// TIA Portal V21 export
DATA_BLOCK "Paratia"   // DB25
{ S7_Optimized_Access := 'TRUE' }
// stored: MemoryReserve 100
   VAR RETAIN
      P : Array[0.."K_NumParatia"] of "Std_Paratia";
      Posizionamento : Struct
         Paratia : Array[0.."K_NumParatia"] of Struct
            K_Paratia : Int;   // Costante che inidca la paratia
            PosizioneAttuale : Real;   // Posizione attuale della paratia
            Target : Real;   // Quantità che dovrebbe essere gestita
            TargetOld : Real;
            PercentualeDaScarto : Real;   // Percentuale di apertura per compensare lo scarto totale
            PercentualeDaTarget : Real;   // Percentuale di apertura da target
            PercentualeDaGestire : Real;
            OffsetDaPrecedente : Real;   // Posizione offsetta rispetto alla precedente
            Abilitazione : Bool;   // La paratia è abilitata al funzionamento
            StatoAperta : Bool;   // 1 = Aperta 0 = Chiusa
            MassimoProdottoGestibile : Real;
            PulsanteIncrementa_Premuto : Bool;
            PulsanteDecrementa_Premuto : Bool;
            PulsanteIncrementa_Precedente : Bool;
            PulsanteDecrementa_Precedente : Bool;
            Richieste : Struct
               PercProdottoRichiesto : Real;
               QuotaTrovata : Int;
            END_STRUCT;
            Diagnostica : Struct
               MassimoValoreApertura : Bool;
               ParatiaForzataChiusa : Bool;
               TermicoScattato : Bool;
               OvertimeMovimento : Bool;
               SezionatoreAperto : Bool;
               PresaInCaricoDiExtraProdotto : Bool;
               GestioneScartiDisabilitata : Bool;
               ParatiaDisabilitata : Bool;
               ParatiaNonInAutomatico : Bool;
            END_STRUCT;
            VersoLince : Array[0.."K_NumLinci"] of Struct
               PercorsoAttivo : Bool;
               ProdottoOltreMax : Real;
            END_STRUCT;
         END_STRUCT;
         AbilitazioneGestioneScarti : Bool := TRUE;   // Se abilitato lo scarto viene distribuito tra quelle aperte
         EquidistribuzioneCarico : Bool := FALSE;
         Inizializza : Bool := FALSE;
         PercentualeScartata : Real := 0.0;
         PercentualeGestita : Real := 100.0;
         ProdottoAssegnato : Real := 100.0;
         ProdottoNonAssegnato : Real := 0.0;
         NumeroParatieAperte : Int := 2;
         AbilitazioneCalcoloDistribuzione : Bool := TRUE;
         DistribuzioneProdottoNastro : Struct
            Quota : Array[0..99] of Real;   // Quantità di prodotto per ogni quota
         END_STRUCT;
         TargetAutomatico : Bool := TRUE;
      END_STRUCT;
      ProdottoNecessario : Struct
         Lince : Array[0.."K_NumLinci"] of Struct
            ChiamataProdotto : Bool;
            AlimentataDalleParatie : Bool;
            PercentualeAttuale : Real;   // Livello attuale
            PercentualeMassima : Real;   // Livello massimo gestito
            ProdottoRichiestoAssoluto : Real;   // Tiene conto solo della propria chiamata
            ProdottoRichiestoRelativo : Real;   // Tiene conto anche delle altre paratie in chiamata
            ProdottoRichiestoRelativoConExtra : Real;
            ProdottoRichiestoASorgenti : Real;   // Tiene conto del numero di sorgenti collegate
            NumeroSorgentiAttive : Int;
            MassimoProdottoGestibile : Real;
            ProdottoNonGestibile : Real;
            TotaleProdottoExtraTraSorgenti : Real;
         END_STRUCT;
         TotaleRichiesta : Real := 21.65003;
         ProdottoExtraNonGestito : Real := 0.0;
         TotaleRelativoDiChiPuòGestireExtra : Real := 100.0;
      END_STRUCT;
   END_VAR
   VAR
      Funzioni : Struct
         DefaultPrm : Bool := FALSE;
         TutteInAuto : Bool := FALSE;
         PosizionamentiAutomatici : Bool := TRUE;
         BypassFinecorsa : Bool := FALSE;
         VistaLivelloPrograammatore : Bool := FALSE;
      END_STRUCT;
   END_VAR
BEGIN
   // P[0] : Non usare
   // P[1] : IFT6
   // P[2] : IFT7
   // P[3] : IFT8
   // P[4] : IFT9
   // P[5] : Cubettatrice
   // P[6] : Cernita
   P[0].In.SetpointAuto := 0.0;
   P[1].In.SetpointAuto := 100.0;
   P[2].In.SetpointAuto := 34.0;
   P[3..5].In.SetpointAuto := 0.0;
   P[6].In.SetpointAuto := 40.0;
   P[7..9].In.SetpointAuto := 0.0;
   P[0..9].In.PulsanteIncrementa := FALSE;
   P[0..9].In.PulsanteDecrementa := FALSE;
   P[0..9].In.TermicoIntervenuto := FALSE;
   P[0..9].In.FinecorsaPositivo := FALSE;
   P[0..9].In.FinecorsaNegativo := FALSE;
   P[0].In.AbilitazioneMovimento := FALSE;
   P[1..6].In.AbilitazioneMovimento := TRUE;
   P[7..9].In.AbilitazioneMovimento := FALSE;
   P[0].Prm.IsteresiComando := 10.0;
   P[1..2].Prm.IsteresiComando := 6.5;
   P[3..9].Prm.IsteresiComando := 8.0;
   P[0..9].Prm.AbilitazioneInterpolazione := FALSE;
   P[0].Prm.Interpolazione[0].Setpoint := 0.0;
   P[0].Prm.Interpolazione[1].Setpoint := 20.0;
   P[0].Prm.Interpolazione[2].Setpoint := 40.0;
   P[0].Prm.Interpolazione[3].Setpoint := 60.0;
   P[0].Prm.Interpolazione[4].Setpoint := 80.0;
   P[0].Prm.Interpolazione[5].Setpoint := 100.0;
   P[1].Prm.Interpolazione[0].Setpoint := 0.0;
   P[1].Prm.Interpolazione[1].Setpoint := 20.0;
   P[1].Prm.Interpolazione[2].Setpoint := 40.0;
   P[1].Prm.Interpolazione[3].Setpoint := 60.0;
   P[1].Prm.Interpolazione[4].Setpoint := 80.0;
   P[1].Prm.Interpolazione[5].Setpoint := 100.0;
   P[2].Prm.Interpolazione[0].Setpoint := 0.0;
   P[2].Prm.Interpolazione[1].Setpoint := 20.0;
   P[2].Prm.Interpolazione[2].Setpoint := 40.0;
   P[2].Prm.Interpolazione[3].Setpoint := 60.0;
   P[2].Prm.Interpolazione[4].Setpoint := 80.0;
   P[2].Prm.Interpolazione[5].Setpoint := 100.0;
   P[3].Prm.Interpolazione[0].Setpoint := 0.0;
   P[3].Prm.Interpolazione[1].Setpoint := 20.0;
   P[3].Prm.Interpolazione[2].Setpoint := 40.0;
   P[3].Prm.Interpolazione[3].Setpoint := 60.0;
   P[3].Prm.Interpolazione[4].Setpoint := 80.0;
   P[3].Prm.Interpolazione[5].Setpoint := 100.0;
   P[4].Prm.Interpolazione[0].Setpoint := 0.0;
   P[4].Prm.Interpolazione[1].Setpoint := 20.0;
   P[4].Prm.Interpolazione[2].Setpoint := 40.0;
   P[4].Prm.Interpolazione[3].Setpoint := 60.0;
   P[4].Prm.Interpolazione[4].Setpoint := 80.0;
   P[4].Prm.Interpolazione[5].Setpoint := 100.0;
   P[5].Prm.Interpolazione[0].Setpoint := 0.0;
   P[5].Prm.Interpolazione[1].Setpoint := 20.0;
   P[5].Prm.Interpolazione[2].Setpoint := 40.0;
   P[5].Prm.Interpolazione[3].Setpoint := 60.0;
   P[5].Prm.Interpolazione[4].Setpoint := 80.0;
   P[5].Prm.Interpolazione[5].Setpoint := 100.0;
   P[6].Prm.Interpolazione[0].Setpoint := 0.0;
   P[6].Prm.Interpolazione[1].Setpoint := 20.0;
   P[6].Prm.Interpolazione[2].Setpoint := 40.0;
   P[6].Prm.Interpolazione[3].Setpoint := 60.0;
   P[6].Prm.Interpolazione[4].Setpoint := 80.0;
   P[6].Prm.Interpolazione[5].Setpoint := 100.0;
   P[7].Prm.Interpolazione[0].Setpoint := 0.0;
   P[7].Prm.Interpolazione[1].Setpoint := 20.0;
   P[7].Prm.Interpolazione[2].Setpoint := 40.0;
   P[7].Prm.Interpolazione[3].Setpoint := 60.0;
   P[7].Prm.Interpolazione[4].Setpoint := 80.0;
   P[7].Prm.Interpolazione[5].Setpoint := 100.0;
   P[8].Prm.Interpolazione[0].Setpoint := 0.0;
   P[8].Prm.Interpolazione[1].Setpoint := 20.0;
   P[8].Prm.Interpolazione[2].Setpoint := 40.0;
   P[8].Prm.Interpolazione[3].Setpoint := 60.0;
   P[8].Prm.Interpolazione[4].Setpoint := 80.0;
   P[8].Prm.Interpolazione[5].Setpoint := 100.0;
   P[9].Prm.Interpolazione[0].Setpoint := 0.0;
   P[9].Prm.Interpolazione[1].Setpoint := 20.0;
   P[9].Prm.Interpolazione[2].Setpoint := 40.0;
   P[9].Prm.Interpolazione[3].Setpoint := 60.0;
   P[9].Prm.Interpolazione[4].Setpoint := 80.0;
   P[9].Prm.Interpolazione[5].Setpoint := 100.0;
   P[0].Prm.Interpolazione[0].Valore := 0.0;
   P[0].Prm.Interpolazione[1].Valore := 20.0;
   P[0].Prm.Interpolazione[2].Valore := 40.0;
   P[0].Prm.Interpolazione[3].Valore := 60.0;
   P[0].Prm.Interpolazione[4].Valore := 80.0;
   P[0].Prm.Interpolazione[5].Valore := 100.0;
   P[1].Prm.Interpolazione[0].Valore := 0.0;
   P[1].Prm.Interpolazione[1].Valore := 20.0;
   P[1].Prm.Interpolazione[2].Valore := 40.0;
   P[1].Prm.Interpolazione[3].Valore := 60.0;
   P[1].Prm.Interpolazione[4].Valore := 80.0;
   P[1].Prm.Interpolazione[5].Valore := 100.0;
   P[2].Prm.Interpolazione[0].Valore := 0.0;
   P[2].Prm.Interpolazione[1].Valore := 20.0;
   P[2].Prm.Interpolazione[2].Valore := 40.0;
   P[2].Prm.Interpolazione[3].Valore := 60.0;
   P[2].Prm.Interpolazione[4].Valore := 80.0;
   P[2].Prm.Interpolazione[5].Valore := 100.0;
   P[3].Prm.Interpolazione[0].Valore := 0.0;
   P[3].Prm.Interpolazione[1].Valore := 20.0;
   P[3].Prm.Interpolazione[2].Valore := 40.0;
   P[3].Prm.Interpolazione[3].Valore := 60.0;
   P[3].Prm.Interpolazione[4].Valore := 80.0;
   P[3].Prm.Interpolazione[5].Valore := 100.0;
   P[4].Prm.Interpolazione[0].Valore := 0.0;
   P[4].Prm.Interpolazione[1].Valore := 20.0;
   P[4].Prm.Interpolazione[2].Valore := 40.0;
   P[4].Prm.Interpolazione[3].Valore := 60.0;
   P[4].Prm.Interpolazione[4].Valore := 80.0;
   P[4].Prm.Interpolazione[5].Valore := 100.0;
   P[5].Prm.Interpolazione[0].Valore := 0.0;
   P[5].Prm.Interpolazione[1].Valore := 20.0;
   P[5].Prm.Interpolazione[2].Valore := 40.0;
   P[5].Prm.Interpolazione[3].Valore := 60.0;
   P[5].Prm.Interpolazione[4].Valore := 80.0;
   P[5].Prm.Interpolazione[5].Valore := 100.0;
   P[6].Prm.Interpolazione[0].Valore := 0.0;
   P[6].Prm.Interpolazione[1].Valore := 20.0;
   P[6].Prm.Interpolazione[2].Valore := 40.0;
   P[6].Prm.Interpolazione[3].Valore := 60.0;
   P[6].Prm.Interpolazione[4].Valore := 80.0;
   P[6].Prm.Interpolazione[5].Valore := 100.0;
   P[7].Prm.Interpolazione[0].Valore := 0.0;
   P[7].Prm.Interpolazione[1].Valore := 20.0;
   P[7].Prm.Interpolazione[2].Valore := 40.0;
   P[7].Prm.Interpolazione[3].Valore := 60.0;
   P[7].Prm.Interpolazione[4].Valore := 80.0;
   P[7].Prm.Interpolazione[5].Valore := 100.0;
   P[8].Prm.Interpolazione[0].Valore := 0.0;
   P[8].Prm.Interpolazione[1].Valore := 20.0;
   P[8].Prm.Interpolazione[2].Valore := 40.0;
   P[8].Prm.Interpolazione[3].Valore := 60.0;
   P[8].Prm.Interpolazione[4].Valore := 80.0;
   P[8].Prm.Interpolazione[5].Valore := 100.0;
   P[9].Prm.Interpolazione[0].Valore := 0.0;
   P[9].Prm.Interpolazione[1].Valore := 20.0;
   P[9].Prm.Interpolazione[2].Valore := 40.0;
   P[9].Prm.Interpolazione[3].Valore := 60.0;
   P[9].Prm.Interpolazione[4].Valore := 80.0;
   P[9].Prm.Interpolazione[5].Valore := 100.0;
   P[0].Dati.AnalogicaReale := 0.0;
   P[1].Dati.AnalogicaReale := 101.2339;
   P[2].Dati.AnalogicaReale := 34.72675;
   P[3].Dati.AnalogicaReale := 0.0;
   P[4].Dati.AnalogicaReale := 0.4089539;
   P[5].Dati.AnalogicaReale := 0.0;
   P[6].Dati.AnalogicaReale := 45.57193;
   P[7..9].Dati.AnalogicaReale := 0.0;
   P[0].Dati.PosizioneAttuale := 0.0;
   P[1].Dati.PosizioneAttuale := 101.2339;
   P[2].Dati.PosizioneAttuale := 34.72675;
   P[3].Dati.PosizioneAttuale := 0.0;
   P[4].Dati.PosizioneAttuale := 0.4089539;
   P[5].Dati.PosizioneAttuale := 0.0;
   P[6].Dati.PosizioneAttuale := 45.57193;
   P[7..9].Dati.PosizioneAttuale := 0.0;
   P[0].Dati.IncrementaUscita := TRUE;
   P[1..9].Dati.IncrementaUscita := FALSE;
   P[0].Dati.PosizionePrecedente := 0.0;
   P[1].Dati.PosizionePrecedente := 101.0646;
   P[2].Dati.PosizionePrecedente := 24.01413;
   P[3].Dati.PosizionePrecedente := 0.0;
   P[4].Dati.PosizionePrecedente := 10.76733;
   P[5].Dati.PosizionePrecedente := 13.94059;
   P[6].Dati.PosizionePrecedente := 49.32968;
   P[7..9].Dati.PosizionePrecedente := 0.0;
   P[0].Dati.DeltaMovimentoTotale := 0.0;
   P[1].Dati.DeltaMovimentoTotale := 38.55846;
   P[2].Dati.DeltaMovimentoTotale := 95655.14;
   P[3].Dati.DeltaMovimentoTotale := 0.0;
   P[4].Dati.DeltaMovimentoTotale := 276.431;
   P[5].Dati.DeltaMovimentoTotale := 1529.73;
   P[6].Dati.DeltaMovimentoTotale := 26.6803;
   P[7..9].Dati.DeltaMovimentoTotale := 0.0;
   P[0].Dati.DeltaMovimentoTotalePrecedente := 0.0;
   P[1].Dati.DeltaMovimentoTotalePrecedente := 96.96799;
   P[2].Dati.DeltaMovimentoTotalePrecedente := 84.48998;
   P[3].Dati.DeltaMovimentoTotalePrecedente := 0.0;
   P[4].Dati.DeltaMovimentoTotalePrecedente := 6.2173;
   P[5].Dati.DeltaMovimentoTotalePrecedente := 10887.7;
   P[6].Dati.DeltaMovimentoTotalePrecedente := 66.14905;
   P[7..9].Dati.DeltaMovimentoTotalePrecedente := 0.0;
   P[0..9].Dati.VerificaOvertime := FALSE;
   P[0..9].Dati.InAllarme := FALSE;
   P[0..2].Dati.ForzataChiusa := FALSE;
   P[3..4].Dati.ForzataChiusa := TRUE;
   P[5..9].Dati.ForzataChiusa := FALSE;
   P[0..9].Hmi.Auto := TRUE;
   P[0..9].Hmi.Man := FALSE;
   P[0..9].Hmi.PulsanteIncrementa := FALSE;
   P[0..9].Hmi.PulsanteDecrementa := FALSE;
   P[0..9].Hmi.Simulazione := FALSE;
   P[0].Hmi.SetpointBloccato := FALSE;
   P[1..5].Hmi.SetpointBloccato := TRUE;
   P[6..9].Hmi.SetpointBloccato := FALSE;
   P[0..9].Allarmi.TimerRitMov.IN := FALSE;
   P[0..9].Allarmi.TimerRitMov.O := FALSE;
   P[0..9].Allarmi.TimerRitMov.Preset := 5.0;
   P[0..9].Allarmi.TimerRitMov.TempoTrascorso := 0.0;
   P[0..9].Allarmi.PresetSoglie.MinimoSpostamento := 5.0;
   P[0].Allarmi."A"[0..3].Abilitato := FALSE;
   P[1].Allarmi."A"[0..3].Abilitato := FALSE;
   P[2].Allarmi."A"[0..3].Abilitato := FALSE;
   P[3].Allarmi."A"[0..3].Abilitato := FALSE;
   P[4].Allarmi."A"[0..3].Abilitato := FALSE;
   P[5].Allarmi."A"[0..3].Abilitato := FALSE;
   P[6].Allarmi."A"[0..3].Abilitato := FALSE;
   P[7].Allarmi."A"[0..3].Abilitato := FALSE;
   P[8].Allarmi."A"[0..3].Abilitato := FALSE;
   P[9].Allarmi."A"[0..3].Abilitato := FALSE;
   P[0].Allarmi."A"[0..3].Stato := FALSE;
   P[1].Allarmi."A"[0..3].Stato := FALSE;
   P[2].Allarmi."A"[0..3].Stato := FALSE;
   P[3].Allarmi."A"[0..3].Stato := FALSE;
   P[4].Allarmi."A"[0..3].Stato := FALSE;
   P[5].Allarmi."A"[0..3].Stato := FALSE;
   P[6].Allarmi."A"[0..3].Stato := FALSE;
   P[7].Allarmi."A"[0..3].Stato := FALSE;
   P[8].Allarmi."A"[0..3].Stato := FALSE;
   P[9].Allarmi."A"[0..3].Stato := FALSE;
   P[0].Allarmi."A"[0..3].Silenziato := FALSE;
   P[1].Allarmi."A"[0..3].Silenziato := FALSE;
   P[2].Allarmi."A"[0..3].Silenziato := FALSE;
   P[3].Allarmi."A"[0..3].Silenziato := FALSE;
   P[4].Allarmi."A"[0..3].Silenziato := FALSE;
   P[5].Allarmi."A"[0..3].Silenziato := FALSE;
   P[6].Allarmi."A"[0..3].Silenziato := FALSE;
   P[7].Allarmi."A"[0..3].Silenziato := FALSE;
   P[8].Allarmi."A"[0..3].Silenziato := FALSE;
   P[9].Allarmi."A"[0..3].Silenziato := FALSE;
   P[0].Allarmi."A"[0..3].EnWarnHmi := FALSE;
   P[1].Allarmi."A"[0..3].EnWarnHmi := FALSE;
   P[2].Allarmi."A"[0..3].EnWarnHmi := FALSE;
   P[3].Allarmi."A"[0..3].EnWarnHmi := FALSE;
   P[4].Allarmi."A"[0..3].EnWarnHmi := FALSE;
   P[5].Allarmi."A"[0..3].EnWarnHmi := FALSE;
   P[6].Allarmi."A"[0..3].EnWarnHmi := FALSE;
   P[7].Allarmi."A"[0..3].EnWarnHmi := FALSE;
   P[8].Allarmi."A"[0..3].EnWarnHmi := FALSE;
   P[9].Allarmi."A"[0..3].EnWarnHmi := FALSE;
   P[0].Allarmi."A"[0..3].EnCadutaCiclo := FALSE;
   P[1].Allarmi."A"[0..3].EnCadutaCiclo := FALSE;
   P[2].Allarmi."A"[0..3].EnCadutaCiclo := FALSE;
   P[3].Allarmi."A"[0..3].EnCadutaCiclo := FALSE;
   P[4].Allarmi."A"[0..3].EnCadutaCiclo := FALSE;
   P[5].Allarmi."A"[0..3].EnCadutaCiclo := FALSE;
   P[6].Allarmi."A"[0..3].EnCadutaCiclo := FALSE;
   P[7].Allarmi."A"[0..3].EnCadutaCiclo := FALSE;
   P[8].Allarmi."A"[0..3].EnCadutaCiclo := FALSE;
   P[9].Allarmi."A"[0..3].EnCadutaCiclo := FALSE;
   P[0..9].Allarmi.WordHMI := 16#0000;
   P[0..9].Out.CmdPos := FALSE;
   P[0..9].Out.CmdNeg := FALSE;
   P[0].Rif_Inc.K_AnalogicaPosAttuale := 0;
   P[1].Rif_Inc.K_AnalogicaPosAttuale := 76;
   P[2].Rif_Inc.K_AnalogicaPosAttuale := 75;
   P[3].Rif_Inc.K_AnalogicaPosAttuale := 0;
   P[4].Rif_Inc.K_AnalogicaPosAttuale := 73;
   P[5].Rif_Inc.K_AnalogicaPosAttuale := 74;
   P[6].Rif_Inc.K_AnalogicaPosAttuale := 67;
   P[7..9].Rif_Inc.K_AnalogicaPosAttuale := 0;
   P[0..9].Rif_Inc.K_AnalogicaRiferimento := 0;
   P[0..9].Rif_Inc.K_StazioneRiferimento := 0;
   Posizionamento.Paratia[0].K_Paratia := 0;
   Posizionamento.Paratia[1].K_Paratia := 5;
   Posizionamento.Paratia[2].K_Paratia := 4;
   Posizionamento.Paratia[3].K_Paratia := 3;
   Posizionamento.Paratia[4].K_Paratia := 2;
   Posizionamento.Paratia[5].K_Paratia := 1;
   Posizionamento.Paratia[6..9].K_Paratia := 0;
   Posizionamento.Paratia[0..1].PosizioneAttuale := 0.0;
   Posizionamento.Paratia[2].PosizioneAttuale := 0.4089539;
   Posizionamento.Paratia[3].PosizioneAttuale := 0.0;
   Posizionamento.Paratia[4].PosizioneAttuale := 34.72675;
   Posizionamento.Paratia[5].PosizioneAttuale := 101.2339;
   Posizionamento.Paratia[6..9].PosizioneAttuale := 0.0;
   Posizionamento.Paratia[0].Target := 25.0;
   Posizionamento.Paratia[1..3].Target := 0.0;
   Posizionamento.Paratia[4].Target := 60.0;
   Posizionamento.Paratia[5].Target := 40.0;
   Posizionamento.Paratia[6..9].Target := 25.0;
   Posizionamento.Paratia[0..3].TargetOld := 0.0;
   Posizionamento.Paratia[4].TargetOld := 60.0;
   Posizionamento.Paratia[5].TargetOld := 40.0;
   Posizionamento.Paratia[6..9].TargetOld := 0.0;
   Posizionamento.Paratia[0..9].PercentualeDaScarto := 0.0;
   Posizionamento.Paratia[0..3].PercentualeDaTarget := 0.0;
   Posizionamento.Paratia[4].PercentualeDaTarget := 60.0;
   Posizionamento.Paratia[5].PercentualeDaTarget := 40.0;
   Posizionamento.Paratia[6..9].PercentualeDaTarget := 0.0;
   Posizionamento.Paratia[0..3].PercentualeDaGestire := 0.0;
   Posizionamento.Paratia[4].PercentualeDaGestire := 60.0;
   Posizionamento.Paratia[5].PercentualeDaGestire := 40.0;
   Posizionamento.Paratia[6..9].PercentualeDaGestire := 0.0;
   Posizionamento.Paratia[0..4].OffsetDaPrecedente := 0.0;
   Posizionamento.Paratia[5].OffsetDaPrecedente := 60.0;
   Posizionamento.Paratia[6..9].OffsetDaPrecedente := 0.0;
   Posizionamento.Paratia[0].Abilitazione := FALSE;
   Posizionamento.Paratia[1..2].Abilitazione := TRUE;
   Posizionamento.Paratia[3].Abilitazione := FALSE;
   Posizionamento.Paratia[4..5].Abilitazione := TRUE;
   Posizionamento.Paratia[6..9].Abilitazione := FALSE;
   Posizionamento.Paratia[0..3].StatoAperta := FALSE;
   Posizionamento.Paratia[4..5].StatoAperta := TRUE;
   Posizionamento.Paratia[6..9].StatoAperta := FALSE;
   Posizionamento.Paratia[0].MassimoProdottoGestibile := 100.0;
   Posizionamento.Paratia[1..2].MassimoProdottoGestibile := 40.0;
   Posizionamento.Paratia[3].MassimoProdottoGestibile := 0.0;
   Posizionamento.Paratia[4].MassimoProdottoGestibile := 60.0;
   Posizionamento.Paratia[5].MassimoProdottoGestibile := 40.0;
   Posizionamento.Paratia[6..9].MassimoProdottoGestibile := 100.0;
   Posizionamento.Paratia[0..9].PulsanteIncrementa_Premuto := FALSE;
   Posizionamento.Paratia[0..9].PulsanteDecrementa_Premuto := FALSE;
   Posizionamento.Paratia[0..9].PulsanteIncrementa_Precedente := FALSE;
   Posizionamento.Paratia[0..9].PulsanteDecrementa_Precedente := FALSE;
   Posizionamento.Paratia[0..3].Richieste.PercProdottoRichiesto := 0.0;
   Posizionamento.Paratia[4].Richieste.PercProdottoRichiesto := 60.0;
   Posizionamento.Paratia[5].Richieste.PercProdottoRichiesto := 40.0;
   Posizionamento.Paratia[6..9].Richieste.PercProdottoRichiesto := 0.0;
   Posizionamento.Paratia[0..3].Richieste.QuotaTrovata := 0;
   Posizionamento.Paratia[4].Richieste.QuotaTrovata := 34;
   Posizionamento.Paratia[5].Richieste.QuotaTrovata := 100;
   Posizionamento.Paratia[6..9].Richieste.QuotaTrovata := 0;
   Posizionamento.Paratia[0..9].Diagnostica.MassimoValoreApertura := FALSE;
   Posizionamento.Paratia[0].Diagnostica.ParatiaForzataChiusa := FALSE;
   Posizionamento.Paratia[1..3].Diagnostica.ParatiaForzataChiusa := TRUE;
   Posizionamento.Paratia[4..9].Diagnostica.ParatiaForzataChiusa := FALSE;
   Posizionamento.Paratia[0..9].Diagnostica.TermicoScattato := FALSE;
   Posizionamento.Paratia[0..9].Diagnostica.OvertimeMovimento := FALSE;
   Posizionamento.Paratia[0..9].Diagnostica.SezionatoreAperto := FALSE;
   Posizionamento.Paratia[0..9].Diagnostica.PresaInCaricoDiExtraProdotto := FALSE;
   Posizionamento.Paratia[0..9].Diagnostica.GestioneScartiDisabilitata := FALSE;
   Posizionamento.Paratia[0..2].Diagnostica.ParatiaDisabilitata := FALSE;
   Posizionamento.Paratia[3].Diagnostica.ParatiaDisabilitata := TRUE;
   Posizionamento.Paratia[4..9].Diagnostica.ParatiaDisabilitata := FALSE;
   Posizionamento.Paratia[0..9].Diagnostica.ParatiaNonInAutomatico := FALSE;
   Posizionamento.Paratia[0].VersoLince[0..4].PercorsoAttivo := FALSE;
   Posizionamento.Paratia[1].VersoLince[0..4].PercorsoAttivo := FALSE;
   Posizionamento.Paratia[2].VersoLince[0..4].PercorsoAttivo := FALSE;
   Posizionamento.Paratia[3].VersoLince[0..4].PercorsoAttivo := FALSE;
   Posizionamento.Paratia[4].VersoLince[0..2].PercorsoAttivo := FALSE;
   Posizionamento.Paratia[4].VersoLince[3].PercorsoAttivo := TRUE;
   Posizionamento.Paratia[4].VersoLince[4].PercorsoAttivo := FALSE;
   Posizionamento.Paratia[5].VersoLince[0..2].PercorsoAttivo := FALSE;
   Posizionamento.Paratia[5].VersoLince[3].PercorsoAttivo := TRUE;
   Posizionamento.Paratia[5].VersoLince[4].PercorsoAttivo := FALSE;
   Posizionamento.Paratia[6].VersoLince[0..4].PercorsoAttivo := FALSE;
   Posizionamento.Paratia[7].VersoLince[0..4].PercorsoAttivo := FALSE;
   Posizionamento.Paratia[8].VersoLince[0..4].PercorsoAttivo := FALSE;
   Posizionamento.Paratia[9].VersoLince[0..4].PercorsoAttivo := FALSE;
   Posizionamento.Paratia[0].VersoLince[0..4].ProdottoOltreMax := 0.0;
   Posizionamento.Paratia[1].VersoLince[0..4].ProdottoOltreMax := 0.0;
   Posizionamento.Paratia[2].VersoLince[0..4].ProdottoOltreMax := 0.0;
   Posizionamento.Paratia[3].VersoLince[0..4].ProdottoOltreMax := 0.0;
   Posizionamento.Paratia[4].VersoLince[0..4].ProdottoOltreMax := 0.0;
   Posizionamento.Paratia[5].VersoLince[0..2].ProdottoOltreMax := 0.0;
   Posizionamento.Paratia[5].VersoLince[3].ProdottoOltreMax := 10.0;
   Posizionamento.Paratia[5].VersoLince[4].ProdottoOltreMax := 0.0;
   Posizionamento.Paratia[6].VersoLince[0..4].ProdottoOltreMax := 0.0;
   Posizionamento.Paratia[7].VersoLince[0..4].ProdottoOltreMax := 0.0;
   Posizionamento.Paratia[8].VersoLince[0..4].ProdottoOltreMax := 0.0;
   Posizionamento.Paratia[9].VersoLince[0..4].ProdottoOltreMax := 0.0;
   // Posizionamento.Paratia[0] : Non usare
   // Posizionamento.Paratia[1] : Cubettatrice
   // Posizionamento.Paratia[2] : IFT8
   // Posizionamento.Paratia[3] : IFT9
   // Posizionamento.Paratia[4] : IFT7
   // Posizionamento.Paratia[5] : IFT6
   Posizionamento.DistribuzioneProdottoNastro.Quota[0..5] := 10.0;
   Posizionamento.DistribuzioneProdottoNastro.Quota[6..25] := 25.0;
   Posizionamento.DistribuzioneProdottoNastro.Quota[26..35] := 35.0;
   Posizionamento.DistribuzioneProdottoNastro.Quota[36..60] := 15.0;
   Posizionamento.DistribuzioneProdottoNastro.Quota[61..70] := 5.0;
   Posizionamento.DistribuzioneProdottoNastro.Quota[71..99] := 1.0;
   ProdottoNecessario.Lince[0..2].ChiamataProdotto := FALSE;
   ProdottoNecessario.Lince[3].ChiamataProdotto := TRUE;
   ProdottoNecessario.Lince[4].ChiamataProdotto := FALSE;
   ProdottoNecessario.Lince[0..2].AlimentataDalleParatie := FALSE;
   ProdottoNecessario.Lince[3].AlimentataDalleParatie := TRUE;
   ProdottoNecessario.Lince[4].AlimentataDalleParatie := FALSE;
   ProdottoNecessario.Lince[0].PercentualeAttuale := 0.0;
   ProdottoNecessario.Lince[1].PercentualeAttuale := 58.03829;
   ProdottoNecessario.Lince[2].PercentualeAttuale := 0.003985969;
   ProdottoNecessario.Lince[3].PercentualeAttuale := 38.34997;
   ProdottoNecessario.Lince[4].PercentualeAttuale := 0.0;
   ProdottoNecessario.Lince[0].PercentualeMassima := 0.0;
   ProdottoNecessario.Lince[1].PercentualeMassima := 55.0;
   ProdottoNecessario.Lince[2].PercentualeMassima := 70.0;
   ProdottoNecessario.Lince[3].PercentualeMassima := 60.0;
   ProdottoNecessario.Lince[4].PercentualeMassima := 0.0;
   ProdottoNecessario.Lince[0..2].ProdottoRichiestoAssoluto := 0.0;
   ProdottoNecessario.Lince[3].ProdottoRichiestoAssoluto := 21.65003;
   ProdottoNecessario.Lince[4].ProdottoRichiestoAssoluto := 0.0;
   ProdottoNecessario.Lince[0..2].ProdottoRichiestoRelativo := 0.0;
   ProdottoNecessario.Lince[3].ProdottoRichiestoRelativo := 100.0;
   ProdottoNecessario.Lince[4].ProdottoRichiestoRelativo := 0.0;
   ProdottoNecessario.Lince[0..2].ProdottoRichiestoRelativoConExtra := 0.0;
   ProdottoNecessario.Lince[3].ProdottoRichiestoRelativoConExtra := 100.0;
   ProdottoNecessario.Lince[4].ProdottoRichiestoRelativoConExtra := 0.0;
   ProdottoNecessario.Lince[0..2].ProdottoRichiestoASorgenti := 0.0;
   ProdottoNecessario.Lince[3].ProdottoRichiestoASorgenti := 50.0;
   ProdottoNecessario.Lince[4].ProdottoRichiestoASorgenti := 0.0;
   ProdottoNecessario.Lince[0..2].NumeroSorgentiAttive := 0;
   ProdottoNecessario.Lince[3].NumeroSorgentiAttive := 2;
   ProdottoNecessario.Lince[4].NumeroSorgentiAttive := 0;
   ProdottoNecessario.Lince[0..2].MassimoProdottoGestibile := 0.0;
   ProdottoNecessario.Lince[3].MassimoProdottoGestibile := 100.0;
   ProdottoNecessario.Lince[4].MassimoProdottoGestibile := 0.0;
   ProdottoNecessario.Lince[0..4].ProdottoNonGestibile := 0.0;
   ProdottoNecessario.Lince[0..2].TotaleProdottoExtraTraSorgenti := 0.0;
   ProdottoNecessario.Lince[3].TotaleProdottoExtraTraSorgenti := 10.0;
   ProdottoNecessario.Lince[4].TotaleProdottoExtraTraSorgenti := 0.0;
   // ProdottoNecessario.Lince[1] : Lince 1
   // ProdottoNecessario.Lince[2] : Lince 2
   // ProdottoNecessario.Lince[3] : Lince 3
END_DATA_BLOCK
